Staubli VAL3: insertInstr.pgx

program insertInstr(string& x_sItem[])
  local num i
  local num l_nNum
begin
  // TODO
  call use:setSizeList(14,0,10,11)
  call use:setView(false)
  call use:listcreate("Select")
  // insert the action on Point

  call use:listupdate(0)
  // SELECT THE ITEM
  x_sItem=""
  do
    i=getKey()
    l_nNum=0
    call use:listevent(i,l_nNum,x_sItem)
    delay(0)
  until i==255 or i==270
  //

  // NOT GOOD
  x_sItem=""
end
